FUNCTION_BLOCK FB_KillMultipleNavigationPS
VAR_INPUT
	Ps	: POINTER TO BOOL;
END_VAR
VAR
	i : USINT;
	activeCount : UINT;
	TON_DelayResetPs : TON;
END_VAR

activeCount := 0;
FOR i := 0 TO 20 DO
    IF Ps[i] THEN
        activeCount := activeCount + 1;
    END_IF
END_FOR

TON_DelayResetPs(IN := activeCount > 1, PT := T#500MS);

IF TON_DelayResetPs.Q THEN
	MEMSET(Ps, 0, SIZEOF(HMI.In.Navigation.PS)-SIZEOF(BOOL));
	activeCount := 0;
END_IF

END_FUNCTION_BLOCK

(* stored: Version 1.1.0.1, ProductVersion 3.1.4024.15
   POU FB_KillMultipleNavigationPS: Id {5c5d6d24-93f0-4d59-8e11-f1f0e7ebc027}, SpecialFunc None *)
